TYPE DUT_SENSOR_DATAS_2 :
UNION
	data_lreal:REAL;
	data_byte:ARRAY[0..3] OF BYTE;
END_UNION
END_TYPE

(* stored: Version 1.1.0.1, ProductVersion 3.1.4024.6
   DUT DUT_SENSOR_DATAS_2: Id {9c7e8f95-d554-4f15-bf66-960604e88307} *)
